(* IEC 61131-3 sources: horner-cscape-mcp/examples/st_samples, 4 files *)

(* ---- motor_controller.st ---- *)
(* ============================================================================
 * Title:       FB_MotorController
 * Author:      Horner Cscape MCP Specialist
 * Description:
 *   Industrial DOL & VFD Motor Controller Function Block.
 *   Features:
 *     - E-Stop and Guard Door Safety Interlocks
 *     - Thermal Overload Relay Trip Monitoring (NC)
 *     - Momentary Start (NO) and Stop (NC) Pushbutton Inputs
 *     - Run Feedback (Auxiliary Contactor) Verification with 3.0s Debounce
 *     - Latched Fault Detection with Dedicated Reset Command
 *     - VFD Speed Reference Clamping and Linear Acceleration Ramp
 *     - Retentive Non-Volatile Operating Run Hours Accumulator
 * Target:      Horner OCS / Straton K5 IEC 61131-3 Runtime
 * Language:    IEC 61131-3 Structured Text (ST) ONLY
 * ============================================================================ *)

FUNCTION_BLOCK FB_MotorController
VAR_INPUT
    StartCmd : BOOL;            (* Operator Start Pushbutton (NO) *)
    StopCmd : BOOL;             (* Operator Stop Pushbutton (NC) *)
    SafetyInterlock : BOOL;     (* E-Stop & Safety Guard Circuit OK *)
    OverloadTrip : BOOL;        (* Thermal Overload Relay Status (NC contact, TRUE=Trip) *)
    RunFeedback : BOOL;         (* Contactor Auxiliary Run Feedback Contact *)
    ResetCmd : BOOL;            (* Fault Reset Pushbutton *)
    SpeedSetpoint : REAL;       (* Target VFD Speed Reference (0.0 to 100.0 %) *)
    AccelRate : REAL := 5.0;    (* Ramp acceleration (% per second) *)
    CycleTimeSec : REAL := 0.05;(* PLC scan task cycle time (seconds) *)
END_VAR

VAR_OUTPUT
    MotorRun : BOOL := FALSE;       (* Digital Output to Main Contactor Coil *)
    SpeedRefOut : REAL := 0.0;      (* Analog Output: Current Scaled VFD Speed (0-100%) *)
    StatusRunning : BOOL := FALSE;  (* Verified Motor Running State *)
    FaultActive : BOOL := FALSE;    (* Latched Alarm / Fault Status *)
    OverloadAlarm : BOOL := FALSE;  (* Thermal Overload Trip Indicator *)
    FeedbackFault : BOOL := FALSE;  (* Auxiliary Feedback Failure Alarm *)
    RunHours : UDINT := 0;          (* Retentive Total Operating Run Hours *)
END_VAR

VAR
    FeedbackTimer : TON;            (* Debounce timer for feedback confirmation *)
    RunHourTimer : TON;             (* 1-second pulse timer for run hour tracking *)
    SecondAccumulator : UDINT := 0; (* Internal seconds counter *)
    CurrentSpeedRamp : REAL := 0.0; (* Internal speed ramp value *)
END_VAR

(* 1. Safety Interlocks & Thermal Overload Trip *)
IF NOT SafetyInterlock THEN
    MotorRun := FALSE;
    FaultActive := TRUE;
    CurrentSpeedRamp := 0.0;
END_IF;

IF OverloadTrip THEN
    MotorRun := FALSE;
    FaultActive := TRUE;
    OverloadAlarm := TRUE;
    CurrentSpeedRamp := 0.0;
END_IF;

(* 2. Fault Reset Command *)
IF ResetCmd AND NOT OverloadTrip AND SafetyInterlock THEN
    FaultActive := FALSE;
    OverloadAlarm := FALSE;
    FeedbackFault := FALSE;
END_IF;

(* 3. Start / Stop Logic *)
IF NOT FaultActive AND SafetyInterlock THEN
    IF StartCmd AND NOT StopCmd THEN
        MotorRun := TRUE;
    ELSIF StopCmd THEN
        MotorRun := FALSE;
    END_IF;
END_IF;

(* 4. Auxiliary Feedback Confirmation *)
FeedbackTimer(IN := MotorRun, PT := T#3s);
IF FeedbackTimer.Q AND NOT RunFeedback THEN
    MotorRun := FALSE;
    FaultActive := TRUE;
    FeedbackFault := TRUE;
    CurrentSpeedRamp := 0.0;
END_IF;

StatusRunning := MotorRun AND RunFeedback;

(* 5. VFD Speed Acceleration / Deceleration Ramp *)
IF StatusRunning THEN
    IF CurrentSpeedRamp < SpeedSetpoint THEN
        CurrentSpeedRamp := CurrentSpeedRamp + (AccelRate * CycleTimeSec);
        IF CurrentSpeedRamp > SpeedSetpoint THEN
            CurrentSpeedRamp := SpeedSetpoint;
        END_IF;
    ELSIF CurrentSpeedRamp > SpeedSetpoint THEN
        CurrentSpeedRamp := CurrentSpeedRamp - (AccelRate * CycleTimeSec);
        IF CurrentSpeedRamp < SpeedSetpoint THEN
            CurrentSpeedRamp := SpeedSetpoint;
        END_IF;
    END_IF;
ELSE
    CurrentSpeedRamp := 0.0;
END_IF;

SpeedRefOut := LIMIT(0.0, CurrentSpeedRamp, 100.0);

(* 6. Operating Hours Accumulation *)
RunHourTimer(IN := StatusRunning AND NOT RunHourTimer.Q, PT := T#1s);
IF RunHourTimer.Q THEN
    SecondAccumulator := SecondAccumulator + 1;
    IF SecondAccumulator >= 3600 THEN
        RunHours := RunHours + 1;
        SecondAccumulator := 0;
    END_IF;
END_IF;

END_FUNCTION_BLOCK

(* ---- pid_temperature_loop.st ---- *)
(* ============================================================================
 * Title:       FB_TemperaturePID
 * Author:      Horner Cscape MCP Specialist
 * Description:
 *   Industrial Closed-Loop Temperature PID Controller Function Block.
 *   Features:
 *     - Digital 1st-Order Low-Pass Noise Filter on Raw PV
 *     - Proportional-Integral-Derivative Algorithm with Anti-Reset Windup
 *     - Manual Override Mode with Bumpless Transfer on Mode Switch
 *     - Time-Proportional PWM Output for Solid-State Relay / Contactor
 *     - Multi-Level Process Alarms: High-High, High, Low, Low-Low
 * Target:      Horner OCS / Straton K5 IEC 61131-3 Runtime
 * Language:    IEC 61131-3 Structured Text (ST) ONLY
 * ============================================================================ *)

FUNCTION_BLOCK FB_TemperaturePID
VAR_INPUT
    Setpoint : REAL := 120.0;           (* Desired Temperature in Deg C *)
    RawPV : REAL := 25.0;               (* Unfiltered Sensor Measurement *)
    ManualMode : BOOL := FALSE;         (* TRUE = Manual Override, FALSE = Auto PID *)
    ManualOutput : REAL := 0.0;         (* Manual Control Output (0.0 to 100.0 %) *)
    Kp : REAL := 3.2;                   (* Proportional Gain *)
    Ki : REAL := 0.04;                  (* Integral Gain (1 / sec) *)
    Kd : REAL := 0.25;                  (* Derivative Gain (sec) *)
    FilterAlpha : REAL := 0.20;         (* PV Low-Pass Filter Coefficient (0.0 - 1.0) *)
    CycleTimeSec : REAL := 0.1;         (* PID Update Scan Period (seconds) *)
    PwmPeriodSec : REAL := 10.0;        (* Solid-State Relay Cycle Base Period *)
END_VAR

VAR_OUTPUT
    ControlOutput : REAL := 0.0;        (* Calculated Control Action (0.0 to 100.0 %) *)
    FilteredPV : REAL := 25.0;          (* Noise-Filtered Process Temperature *)
    PWM_HeaterOut : BOOL := FALSE;      (* Solid-State Relay Digital Heating Pulse *)
    Error : REAL := 0.0;                (* Current Regulation Error (SP - PV) *)
    AlarmHH : BOOL := FALSE;            (* Critical High-High Temperature Trip *)
    AlarmH : BOOL := FALSE;             (* High Temperature Warning Alarm *)
    AlarmL : BOOL := FALSE;             (* Low Temperature Warning Alarm *)
    AlarmLL : BOOL := FALSE;            (* Critical Low-Low Temperature Alarm *)
END_VAR

VAR
    LastError : REAL := 0.0;            (* Previous Error for Derivative Term *)
    IntegralSum : REAL := 0.0;          (* Accumulated Integral Action *)
    PropTerm : REAL := 0.0;             (* Proportional Term Component *)
    DerivTerm : REAL := 0.0;            (* Derivative Term Component *)
    RawPIDOutput : REAL := 0.0;         (* Unclamped PID Sum *)
    PwmTimerAcc : REAL := 0.0;          (* Internal PWM Period Accumulator *)
END_VAR

(* 1. First-Order Digital Low-Pass Filter on Process Variable *)
FilteredPV := (FilterAlpha * RawPV) + ((1.0 - FilterAlpha) * FilteredPV);

(* 2. Error Calculation *)
Error := Setpoint - FilteredPV;

(* 3. Process Alarm Limits *)
AlarmHH := FilteredPV >= (Setpoint + 25.0);
AlarmH  := FilteredPV >= (Setpoint + 10.0);
AlarmL  := FilteredPV <= (Setpoint - 10.0);
AlarmLL := FilteredPV <= (Setpoint - 25.0);

(* 4. Automatic / Manual Control Computation *)
IF ManualMode OR AlarmHH THEN
    IF AlarmHH THEN
        ControlOutput := 0.0; (* Safety cut-off on critical overtemperature *)
    ELSE
        ControlOutput := LIMIT(0.0, ManualOutput, 100.0);
    END_IF;
    (* Bumpless transfer tracking *)
    IntegralSum := ControlOutput;
    LastError := Error;
ELSE
    (* Proportional Component *)
    PropTerm := Kp * Error;

    (* Integral Component with Anti-Reset Windup Clamping *)
    IntegralSum := IntegralSum + (Ki * Error * CycleTimeSec);
    IntegralSum := LIMIT(0.0, IntegralSum, 100.0);

    (* Derivative Component *)
    DerivTerm := Kd * (Error - LastError) / CycleTimeSec;
    LastError := Error;

    (* Total Control Effort Clamped to [0.0, 100.0] % *)
    RawPIDOutput := PropTerm + IntegralSum + DerivTerm;
    ControlOutput := LIMIT(0.0, RawPIDOutput, 100.0);
END_IF;

(* 5. Time-Proportional PWM Solid-State Relay Generation *)
PwmTimerAcc := PwmTimerAcc + (CycleTimeSec / PwmPeriodSec * 100.0);
IF PwmTimerAcc >= 100.0 THEN
    PwmTimerAcc := 0.0;
END_IF;

PWM_HeaterOut := (PwmTimerAcc < ControlOutput) AND NOT AlarmHH;

END_FUNCTION_BLOCK

(* ---- batch_mixer.st ---- *)
(* ============================================================================
 * Title:       Prog_BatchMixer
 * Author:      Horner Cscape MCP Specialist
 * Description:
 *   Industrial Food & Beverage Recipe Batch Mixing Sequence Program.
 *   Sequencer States:
 *     - State 0:  IDLE / READY: Awaiting Start Command
 *     - State 10: CHARGE WATER: Metering liquid phase to tare weight
 *     - State 20: FEED SYRUP: High-viscosity ingredient feed with slow agitation
 *     - State 30: HIGH SPEED BLEND: Dual-blade homogenizer timed mix
 *     - State 40: COOK / HEAT: Steam jacket heating to reaction temperature
 *     - State 50: HOLD REACTION: Controlled thermal dwell period
 *     - State 60: TRANSFER / DRAIN: Discharging product to holding tanks
 *     - State 70: CIP FLUSH: Clean-in-Place hot spray wash
 *     - State 99: SAFE ABORT: Immediate actuator lockout on interlock trip
 * Target:      Horner OCS / Straton K5 IEC 61131-3 Runtime
 * Language:    IEC 61131-3 Structured Text (ST) ONLY
 * ============================================================================ *)

PROGRAM Prog_BatchMixer
VAR
    (* Operator Commands *)
    StartBatchCmd : BOOL := FALSE;
    AbortBatchCmd : BOOL := FALSE;
    ResetFaultCmd : BOOL := FALSE;
    SkipToCipCmd  : BOOL := FALSE;

    (* Safety & Sensor Inputs *)
    LidInterlockClosed : BOOL := TRUE;
    VesselHighLevel    : BOOL := FALSE;
    LiquidWeightKg     : REAL := 0.0;
    BatchTemperatureC  : REAL := 22.5;

    (* Recipe Setpoints *)
    RecipeWaterKg      : REAL := 600.0;
    RecipeSyrupKg      : REAL := 250.0;
    RecipeTargetTempC  : REAL := 75.0;
    RecipeMixDuration  : TIME := T#3m;
    RecipeHoldDuration : TIME := T#5m;

    (* Actuator Digital Outputs *)
    ValveWaterSupply   : BOOL := FALSE;
    ValveSyrupSupply   : BOOL := FALSE;
    AgitatorLowSpeed   : BOOL := FALSE;
    AgitatorHighSpeed  : BOOL := FALSE;
    ValveSteamJacket   : BOOL := FALSE;
    ValveBottomDrain   : BOOL := FALSE;
    PumpCIPSpray       : BOOL := FALSE;

    (* Status Flags *)
    BatchRunning       : BOOL := FALSE;
    BatchComplete      : BOOL := FALSE;
    SystemInterlockTrip: BOOL := FALSE;

    (* Sequencer State & Timers *)
    CurrentStep        : INT := 0;
    PreviousStep       : INT := -1;
    TimerMixBlend      : TON;
    TimerReactionHold  : TON;
    TimerCIPWash       : TON;
END_VAR

(* 1. Safety Interlock Supervision *)
SystemInterlockTrip := NOT LidInterlockClosed OR VesselHighLevel OR AbortBatchCmd;

IF SystemInterlockTrip AND CurrentStep <> 0 AND CurrentStep <> 99 THEN
    CurrentStep := 99; (* Transition directly to safe shutdown state *)
END_IF;

(* 2. Main Sequencer State Machine *)
CASE CurrentStep OF
    0: (* IDLE State *)
        ValveWaterSupply  := FALSE;
        ValveSyrupSupply  := FALSE;
        AgitatorLowSpeed  := FALSE;
        AgitatorHighSpeed := FALSE;
        ValveSteamJacket  := FALSE;
        ValveBottomDrain  := FALSE;
        PumpCIPSpray      := FALSE;
        BatchRunning      := FALSE;

        IF StartBatchCmd AND NOT SystemInterlockTrip THEN
            BatchComplete := FALSE;
            BatchRunning  := TRUE;
            CurrentStep   := 10; (* Advance to Charge Water *)
        END_IF;

    10: (* CHARGE WATER *)
        ValveWaterSupply := TRUE;
        IF LiquidWeightKg >= RecipeWaterKg THEN
            ValveWaterSupply := FALSE;
            CurrentStep := 20; (* Advance to Feed Syrup *)
        END_IF;

    20: (* FEED SYRUP WITH LOW SPEED MIXING *)
        ValveSyrupSupply := TRUE;
        AgitatorLowSpeed := TRUE;
        IF LiquidWeightKg >= (RecipeWaterKg + RecipeSyrupKg) THEN
            ValveSyrupSupply := FALSE;
            CurrentStep := 30; (* Advance to High Speed Blend *)
        END_IF;

    30: (* HIGH SPEED BLEND *)
        AgitatorLowSpeed  := FALSE;
        AgitatorHighSpeed := TRUE;
        TimerMixBlend(IN := TRUE, PT := RecipeMixDuration);
        IF TimerMixBlend.Q THEN
            TimerMixBlend(IN := FALSE);
            AgitatorHighSpeed := FALSE;
            CurrentStep := 40; (* Advance to Cooking / Heating *)
        END_IF;

    40: (* STEAM JACKET HEATING *)
        AgitatorLowSpeed := TRUE; (* Keep product moving to prevent scorching *)
        ValveSteamJacket := BatchTemperatureC < RecipeTargetTempC;
        IF BatchTemperatureC >= RecipeTargetTempC THEN
            ValveSteamJacket := FALSE;
            CurrentStep := 50; (* Advance to Reaction Dwell *)
        END_IF;

    50: (* REACTION DWELL HOLD *)
        AgitatorLowSpeed := TRUE;
        ValveSteamJacket := BatchTemperatureC < (RecipeTargetTempC - 1.5);
        TimerReactionHold(IN := TRUE, PT := RecipeHoldDuration);
        IF TimerReactionHold.Q THEN
            TimerReactionHold(IN := FALSE);
            ValveSteamJacket := FALSE;
            CurrentStep := 60; (* Advance to Transfer *)
        END_IF;

    60: (* PRODUCT TRANSFER / VESSEL DRAIN *)
        AgitatorLowSpeed := FALSE;
        ValveBottomDrain := TRUE;
        IF LiquidWeightKg <= 8.0 THEN (* Vessel empty tare threshold *)
            ValveBottomDrain := FALSE;
            CurrentStep := 70; (* Advance to CIP Wash *)
        END_IF;

    70: (* CLEAN-IN-PLACE (CIP) SPRAY WASH *)
        PumpCIPSpray     := TRUE;
        ValveBottomDrain := TRUE;
        TimerCIPWash(IN := TRUE, PT := T#90s);
        IF TimerCIPWash.Q THEN
            TimerCIPWash(IN := FALSE);
            PumpCIPSpray     := FALSE;
            ValveBottomDrain := FALSE;
            BatchComplete    := TRUE;
            BatchRunning     := FALSE;
            CurrentStep      := 0; (* Cycle completed, return to IDLE *)
        END_IF;

    99: (* EMERGENCY SAFE ABORT *)
        ValveWaterSupply  := FALSE;
        ValveSyrupSupply  := FALSE;
        AgitatorLowSpeed  := FALSE;
        AgitatorHighSpeed := FALSE;
        ValveSteamJacket  := FALSE;
        ValveBottomDrain  := FALSE;
        PumpCIPSpray      := FALSE;
        BatchRunning      := FALSE;

        IF ResetFaultCmd AND NOT SystemInterlockTrip THEN
            CurrentStep := 0; (* Cleared to IDLE *)
        END_IF;

    ELSE
        CurrentStep := 0;
END_CASE;

END_PROGRAM

(* ---- modbus_io_handler.st ---- *)
(* ============================================================================
 * Title:       Prog_ModbusIOHandler
 * Author:      Horner Cscape MCP Specialist
 * Description:
 *   Industrial Modbus TCP / RTU Remote Telemetry Processor.
 *   Features:
 *     - Watchdog Counter Heartbeat Supervision (2.0s Timeout)
 *     - Multi-Channel Analog Input Demultiplexing from Modbus Registers
 *     - Engineering Unit Conversion from Raw 0-32000 ADC Horner Counts
 *     - 4-20mA Sensor Out-of-Range & Wire-Break Failure Detection
 *     - Safe Fallback Value Substitution on Fieldbus Offline Status
 *     - Diagnostic Status Bitfield Packing for SCADA / HMI Telemetry
 * Target:      Horner OCS / Straton K5 IEC 61131-3 Runtime
 * Language:    IEC 61131-3 Structured Text (ST) ONLY
 * ============================================================================ *)

PROGRAM Prog_ModbusIOHandler
VAR
    (* Raw Modbus Input Registers *)
    ModbusWatchdogCounter : WORD := 0;
    RawModbusRegisters    : ARRAY [1..8] OF WORD;
    ModbusRxErrorCount    : UDINT := 0;

    (* Scaled Engineering Measurements *)
    FlowRateLPM           : REAL := 0.0;    (* 0.0 to 600.0 LPM *)
    DischargePressureBar  : REAL := 0.0;    (* 0.0 to 25.0 Bar *)
    TankLevelPct          : REAL := 0.0;    (* 0.0 to 100.0 % *)
    ConductivityMicroS    : REAL := 0.0;    (* 0.0 to 2000.0 uS/cm *)

    (* Sensor Health Status *)
    SensorFaultFlow       : BOOL := FALSE;
    SensorFaultPressure   : BOOL := FALSE;
    SensorFaultLevel      : BOOL := FALSE;
    SensorFaultConduct    : BOOL := FALSE;

    (* Comm Health Monitoring *)
    LastHeartbeat         : WORD := 0;
    CommTimeoutAlarm      : BOOL := FALSE;
    WatchdogTimer         : TON;

    (* SCADA Diagnostic Word Output *)
    DiagnosticStatusWord  : WORD := 0;
    TotalValidFrames      : UDINT := 0;
END_VAR

(* 1. Remote Drop Heartbeat Verification *)
IF ModbusWatchdogCounter <> LastHeartbeat THEN
    LastHeartbeat := ModbusWatchdogCounter;
    CommTimeoutAlarm := FALSE;
    TotalValidFrames := TotalValidFrames + 1;
END_IF;

WatchdogTimer(IN := NOT CommTimeoutAlarm, PT := T#2s);
IF WatchdogTimer.Q THEN
    CommTimeoutAlarm := TRUE;
    ModbusRxErrorCount := ModbusRxErrorCount + 1;
END_IF;

(* 2. Analog Processing & Wire Break Detection *)
IF NOT CommTimeoutAlarm THEN
    (* Channel 1: Flow Transmitter (4-20mA = 6400 to 32000 counts) *)
    IF RawModbusRegisters[1] < 3200 THEN (* Under 2mA = Wire break *)
        SensorFaultFlow := TRUE;
        FlowRateLPM := 0.0;
    ELSE
        SensorFaultFlow := FALSE;
        FlowRateLPM := (WORD_TO_REAL(RawModbusRegisters[1]) - 6400.0) * 600.0 / 25600.0;
        FlowRateLPM := LIMIT(0.0, FlowRateLPM, 600.0);
    END_IF;

    (* Channel 2: Discharge Pressure (4-20mA = 6400 to 32000 counts) *)
    IF RawModbusRegisters[2] < 3200 THEN
        SensorFaultPressure := TRUE;
        DischargePressureBar := 0.0;
    ELSE
        SensorFaultPressure := FALSE;
        DischargePressureBar := (WORD_TO_REAL(RawModbusRegisters[2]) - 6400.0) * 25.0 / 25600.0;
        DischargePressureBar := LIMIT(0.0, DischargePressureBar, 25.0);
    END_IF;

    (* Channel 3: Tank Hydrostatic Level (0-10V = 0 to 32000 counts) *)
    SensorFaultLevel := RawModbusRegisters[3] > 32500; (* Overvoltage *)
    TankLevelPct := WORD_TO_REAL(RawModbusRegisters[3]) * 100.0 / 32000.0;
    TankLevelPct := LIMIT(0.0, TankLevelPct, 100.0);

    (* Channel 4: Water Conductivity (0-2000 uS/cm) *)
    SensorFaultConduct := RawModbusRegisters[4] < 100;
    ConductivityMicroS := WORD_TO_REAL(RawModbusRegisters[4]) * 2000.0 / 32000.0;
    ConductivityMicroS := LIMIT(0.0, ConductivityMicroS, 2000.0);
ELSE
    (* Fallback failsafe conditions during comm interruption *)
    FlowRateLPM          := 0.0;
    DischargePressureBar := 0.0;
    TankLevelPct         := 0.0;
    ConductivityMicroS   := 0.0;
END_IF;

(* 3. Diagnostic Bitfield Assembly for HMI/SCADA *)
(* Bit 0: Comm OK, Bit 1: Comm Timeout, Bit 2-5: Sensor Faults *)
IF CommTimeoutAlarm THEN
    DiagnosticStatusWord := 16#0002;
ELSE
    DiagnosticStatusWord := 16#0001;
    IF SensorFaultFlow THEN
        DiagnosticStatusWord := DiagnosticStatusWord OR 16#0004;
    END_IF;
    IF SensorFaultPressure THEN
        DiagnosticStatusWord := DiagnosticStatusWord OR 16#0008;
    END_IF;
    IF SensorFaultLevel THEN
        DiagnosticStatusWord := DiagnosticStatusWord OR 16#0010;
    END_IF;
    IF SensorFaultConduct THEN
        DiagnosticStatusWord := DiagnosticStatusWord OR 16#0020;
    END_IF;
END_IF;

END_PROGRAM
